(*

.. <legal notes>

legal notes
=================
| SPDX-FileCopyrightText: © 2026 Oleksandr Tiutyk <trofimich@gmail.com>
| SPDX-License-Identifier: LGPL-3.0-only
| For details check: LGPL-3.0-only_

.. _LGPL-3.0-only: https://www.gnu.org/licenses/lgpl-3.0.en.html

.. </legal notes>

*)

{attribute 'no_explicit_call' := 'do not call this function block directly'} 
FUNCTION_BLOCK SignalControlledIntersectionAutomationController EXTENDS TOF_Automation.AutomationController<7>
VAR CONSTANT
	RED_GREEN_LIGHT_INTERVAL : TIME := T#4000MS;
	YELLOW_LIGHT_INTERVAL : TIME := T#1000MS;
	FLASHING_YELLOW_LIGHT_INTERVAL : TIME := T#800MS;	
	
	SWITCH_SPEED_FACTOR : LREAL := 3; // +/- 30%
END_VAR
VAR_INPUT
	ThrowTestExceptionRequest : BOOL;
	TestExceptionMessage : STRING := 'Test error message';

	ResetRequest : BOOL;
END_VAR
VAR_OUTPUT	
	IntersectionMode : SIGNAL_CONTROLLED_INTERSECTION_MODE;
	IntersectionState : SIGNAL_CONTROLLED_INTERSECTION_STATE;

	{region "Devices"}
	
	WorkingModeSwitch : TOF_Devices_IO.DigitalInput("WorkingModeSwitch", THIS^);
	
	BlinkingYellowModeSwitch : TOF_Devices_IO.DigitalInput("BlinkingYellowModeSwitch", THIS^);
	
	SpeedAdjusterConverter : TOF_Devices_IO.RangeAnalogValueConverter(-20, +20, TOF_Devices_IO.RawAnalogValues.FromInt16(TOF_Core.SignedInt16.MIN_VALUE), TOF_Devices_IO.RawAnalogValues.FromInt16(TOF_Core.SignedInt16.MAX_VALUE));
	SwitchSpeedAdjuster : TOF_Devices_IO.AnalogInput("SwitchSpeedAdjuster", THIS^, SpeedAdjusterConverter);
	
	TrafficLight1 : TrafficLight("TrafficLight1", THIS^);
	TrafficLight2 : TrafficLight("TrafficLight2", THIS^);
	TrafficLight3 : TrafficLight("TrafficLight3", THIS^);
	TrafficLight4 : TrafficLight("TrafficLight4", THIS^);
	
 	{endregion} 	
END_VAR
VAR	
	_ClassName : STRING := __POUNAME();

	_Devices : ARRAY [0.._ChildCount - 1] OF TOF_Automation.IChildAutomationComponent := 
	[
		WorkingModeSwitch, 
		BlinkingYellowModeSwitch, 
		SwitchSpeedAdjuster, 
		TrafficLight1, 
		TrafficLight2, 
		TrafficLight3, 
		TrafficLight4
	];
	
	_OperationalStateChanged : BOOL;
	
	{region "Timers"}
	
	_RedGreenLightTimer : TOF_Timers.Timer;
	_YellowLightTimer : TOF_Timers.Timer;

	_FlashingYellowLightTimer : TOF_Timers.Timer;
	
	{endregion}
END_VAR

METHOD PRIVATE bindIO
WorkingModeSwitch.BindToIO(
	Terminals.DI_1.Channel_1
);

BlinkingYellowModeSwitch.BindToIO(
	Terminals.DI_1.Channel_2
);

SwitchSpeedAdjuster.BindToInt16IO(Terminals.AI_3.Channel_1);

TrafficLight1.BindToIO(
	redLightRawValue 	:= Terminals.DO_2.Channel_1,
	yellowLightRawValue := Terminals.DO_2.Channel_2,
	greenLightRawValue 	:= Terminals.DO_2.Channel_3	
);
TrafficLight2.BindToIO(
	redLightRawValue 	:= Terminals.DO_2.Channel_4,
	yellowLightRawValue := Terminals.DO_2.Channel_5,
	greenLightRawValue 	:= Terminals.DO_2.Channel_6	
);
TrafficLight3.BindToIO(
	redLightRawValue 	:= Terminals.DO_2.Channel_7,
	yellowLightRawValue := Terminals.DO_2.Channel_8,
	greenLightRawValue 	:= Terminals.DO_2.Channel_9	
);
TrafficLight4.BindToIO(
	redLightRawValue 	:= Terminals.DO_2.Channel_10,
	yellowLightRawValue := Terminals.DO_2.Channel_11,
	greenLightRawValue 	:= Terminals.DO_2.Channel_12	
);
END_METHOD

METHOD PRIVATE calculateCorrectedInterval : TIME
VAR_INPUT
	originalInterval : TIME;
	correctionPercent : SINT(-50..50);
END_VAR
IF correctionPercent = 0 THEN
	calculateCorrectedInterval := originalInterval;
ELSIF correctionPercent > 0 THEN
	calculateCorrectedInterval := originalInterval + TO_TIME(TO_INT(originalInterval) * correctionPercent / 100);
ELSE
	calculateCorrectedInterval := originalInterval - TO_TIME(TO_INT(originalInterval) * -correctionPercent / 100);
END_IF
END_METHOD

PROPERTY Children : REFERENCE TO ARRAY [0.._ChildCount - 1] OF TOF_Automation.IChildAutomationComponent
GET
Children REF= _Devices;
END_GET
END_PROPERTY

{attribute 'monitoring' := 'call'}
PROPERTY ClassName : STRING
GET
ClassName := _ClassName;
END_GET
END_PROPERTY

METHOD PRIVATE executeTimers
_RedGreenLightTimer.Execute();
_YellowLightTimer.Execute();
_FlashingYellowLightTimer.Execute();
END_METHOD

{attribute 'monitoring' := 'call'}
PROPERTY NamespaceName : STRING
GET
NamespaceName := CurrentNamespace.Name;
END_GET
END_PROPERTY

METHOD PROTECTED OnBeforeChildrenInitializing
_RedGreenLightTimer.Interval := RED_GREEN_LIGHT_INTERVAL;
_YellowLightTimer.Interval := YELLOW_LIGHT_INTERVAL;

_FlashingYellowLightTimer.Interval := FLASHING_YELLOW_LIGHT_INTERVAL;

bindIO();
END_METHOD

METHOD PROTECTED OnFault
startIdelingMode();

IF ResetRequest THEN
	ResetRequest := FALSE;
	
	Reset();
END_IF
END_METHOD

METHOD PROTECTED OnOperationalStateChanged
VAR_INPUT
	previousState : TOF_Automation.OPERATIONAL_STATE;
END_VAR
_OperationalStateChanged := TRUE;
END_METHOD

METHOD PROTECTED OnWorking
VAR
	testException : TOF_Core.StandardException;
END_VAR
executeTimers();

IF _OperationalStateChanged OR_ELSE WorkingModeSwitch.Changed OR_ELSE BlinkingYellowModeSwitch.Changed THEN
	_OperationalStateChanged := FALSE;
	
	IF NOT WorkingModeSwitch.Value THEN
		startIdelingMode();
	ELSE
		IF BlinkingYellowModeSwitch.Value THEN
			startBlinkingYellowMode();
		ELSE
			startNormalMode();
		END_IF	
	END_IF
	
	RETURN;
ELSE
	CASE IntersectionMode OF
		SIGNAL_CONTROLLED_INTERSECTION_MODE.NORMAL:
			processNormalMode();
		
		SIGNAL_CONTROLLED_INTERSECTION_MODE.BLINKING_YELLOW:
			processBlinkingYellowMode();
	END_CASE
END_IF

IF ThrowTestExceptionRequest THEN
	ThrowTestExceptionRequest := FALSE;
	testException.ThrowByObject(THIS^, __POUNAME(), __POSITION(), TO_WSTRING(TestExceptionMessage), 0);
END_IF
END_METHOD

{attribute 'monitoring' := 'call'}
PROPERTY OperationalStateName : STRING(16)
GET
OperationalStateName := TO_STRING(_OperationalState);
END_GET
END_PROPERTY

METHOD PRIVATE processBlinkingYellowMode
IF _FlashingYellowLightTimer.Elapsed THEN
	IF IntersectionState = SIGNAL_CONTROLLED_INTERSECTION_STATE.ALL_YELLOW THEN
		IntersectionState := SIGNAL_CONTROLLED_INTERSECTION_STATE.ALL_OFF;
	ELSE
		IntersectionState := SIGNAL_CONTROLLED_INTERSECTION_STATE.ALL_YELLOW;
	END_IF
	
	startFlashingYellowLightTimer();
	
	updateTraficLights();
END_IF
END_METHOD

METHOD processNormalMode
CASE IntersectionState OF
	SIGNAL_CONTROLLED_INTERSECTION_STATE._1_3_GREEN_AND_2_4_RED:
		IF _RedGreenLightTimer.Elapsed THEN
			startYellowLightTimer();
			IntersectionState := SIGNAL_CONTROLLED_INTERSECTION_STATE._1_3_YELLOW_AND_2_4_YELLOW;
			updateTraficLights();
		END_IF
 
	SIGNAL_CONTROLLED_INTERSECTION_STATE._1_3_YELLOW_AND_2_4_YELLOW:
		IF _YellowLightTimer.Elapsed THEN
			startRedGreenLightTimer();
			IntersectionState := SIGNAL_CONTROLLED_INTERSECTION_STATE._2_4_GREEN_AND_1_3_RED;
			updateTraficLights();
		END_IF
	
	SIGNAL_CONTROLLED_INTERSECTION_STATE._2_4_GREEN_AND_1_3_RED:
		IF _RedGreenLightTimer.Elapsed THEN
			startYellowLightTimer();
			IntersectionState := SIGNAL_CONTROLLED_INTERSECTION_STATE._2_4_YELLOW_AND_1_3_YELLOW;
			updateTraficLights();
		END_IF
	
	SIGNAL_CONTROLLED_INTERSECTION_STATE._2_4_YELLOW_AND_1_3_YELLOW:
		IF _YellowLightTimer.Elapsed THEN
			startRedGreenLightTimer();
			IntersectionState := SIGNAL_CONTROLLED_INTERSECTION_STATE._1_3_GREEN_AND_2_4_RED;
			updateTraficLights();
		END_IF
	
	ELSE
		startRedGreenLightTimer();
		IntersectionState := SIGNAL_CONTROLLED_INTERSECTION_STATE._1_3_GREEN_AND_2_4_RED;
		updateTraficLights();
END_CASE
END_METHOD

{attribute 'monitoring' := 'call'}
PROPERTY SelfSize : ULINT
GET
SelfSize := XSIZEOF(THIS^);
END_GET
END_PROPERTY

METHOD PRIVATE startBlinkingYellowMode
_RedGreenLightTimer.Cancel();
_YellowLightTimer.Cancel();

startFlashingYellowLightTimer();

IntersectionMode := SIGNAL_CONTROLLED_INTERSECTION_MODE.BLINKING_YELLOW;
IntersectionState := SIGNAL_CONTROLLED_INTERSECTION_STATE.ALL_YELLOW;

updateTraficLights();
END_METHOD

METHOD PRIVATE startFlashingYellowLightTimer
_FlashingYellowLightTimer.Interval := calculateCorrectedInterval(FLASHING_YELLOW_LIGHT_INTERVAL, TO_SINT(SWITCH_SPEED_FACTOR * SwitchSpeedAdjuster.Value));

_FlashingYellowLightTimer.Restart();
END_METHOD

METHOD startIdelingMode
_RedGreenLightTimer.Cancel();
_YellowLightTimer.Cancel();
_FlashingYellowLightTimer.Cancel();

IntersectionMode := SIGNAL_CONTROLLED_INTERSECTION_MODE.IDELING;
IntersectionState := SIGNAL_CONTROLLED_INTERSECTION_STATE.ALL_OFF;

updateTraficLights();
END_METHOD

METHOD startNormalMode
startRedGreenLightTimer();

_YellowLightTimer.Cancel();
_FlashingYellowLightTimer.Cancel();

IntersectionMode := SIGNAL_CONTROLLED_INTERSECTION_MODE.NORMAL;
IntersectionState := SIGNAL_CONTROLLED_INTERSECTION_STATE._1_3_GREEN_AND_2_4_RED;

updateTraficLights();
END_METHOD

METHOD PRIVATE startRedGreenLightTimer
_RedGreenLightTimer.Interval := calculateCorrectedInterval(RED_GREEN_LIGHT_INTERVAL, TO_SINT(SWITCH_SPEED_FACTOR * SwitchSpeedAdjuster.Value));

_RedGreenLightTimer.Restart();
END_METHOD

METHOD PRIVATE startYellowLightTimer
_YellowLightTimer.Interval := calculateCorrectedInterval(YELLOW_LIGHT_INTERVAL, TO_SINT(SWITCH_SPEED_FACTOR * SwitchSpeedAdjuster.Value));

_YellowLightTimer.Restart();
END_METHOD

METHOD PRIVATE updateTraficLights
CASE IntersectionState OF
	SIGNAL_CONTROLLED_INTERSECTION_STATE.ALL_OFF:
		TrafficLight1.SetLight(TRAFFIC_LIGHT_COLOR.NO_COLOR);
		TrafficLight2.SetLight(TRAFFIC_LIGHT_COLOR.NO_COLOR);
		TrafficLight3.SetLight(TRAFFIC_LIGHT_COLOR.NO_COLOR);
		TrafficLight4.SetLight(TRAFFIC_LIGHT_COLOR.NO_COLOR);
	
	SIGNAL_CONTROLLED_INTERSECTION_STATE.ALL_YELLOW, 
	SIGNAL_CONTROLLED_INTERSECTION_STATE._1_3_YELLOW_AND_2_4_YELLOW,
	SIGNAL_CONTROLLED_INTERSECTION_STATE._2_4_YELLOW_AND_1_3_YELLOW:
		TrafficLight1.SetLight(TRAFFIC_LIGHT_COLOR.YELLOW);
		TrafficLight2.SetLight(TRAFFIC_LIGHT_COLOR.YELLOW);
		TrafficLight3.SetLight(TRAFFIC_LIGHT_COLOR.YELLOW);
		TrafficLight4.SetLight(TRAFFIC_LIGHT_COLOR.YELLOW);
	
	SIGNAL_CONTROLLED_INTERSECTION_STATE._1_3_GREEN_AND_2_4_RED:
		TrafficLight1.SetLight(TRAFFIC_LIGHT_COLOR.GREEN);
		TrafficLight2.SetLight(TRAFFIC_LIGHT_COLOR.RED);
		TrafficLight3.SetLight(TRAFFIC_LIGHT_COLOR.GREEN);
		TrafficLight4.SetLight(TRAFFIC_LIGHT_COLOR.RED);
	
	SIGNAL_CONTROLLED_INTERSECTION_STATE._2_4_GREEN_AND_1_3_RED:
		TrafficLight1.SetLight(TRAFFIC_LIGHT_COLOR.RED);
		TrafficLight2.SetLight(TRAFFIC_LIGHT_COLOR.GREEN);
		TrafficLight3.SetLight(TRAFFIC_LIGHT_COLOR.RED);
		TrafficLight4.SetLight(TRAFFIC_LIGHT_COLOR.GREEN);
END_CASE
END_METHOD

END_FUNCTION_BLOCK

(* stored: Version 1.1.0.1
   POU SignalControlledIntersectionAutomationController: Id {d0f0aa39-ea76-461a-8fa3-dba15b8635a6}, SpecialFunc None
   Folder Overriden methods: Id {13702960-9d99-4885-a6ce-63462aae1b07}
   Folder Service methods: Id {856d71ee-39f1-4125-9914-d1908aaa9de4}
   Folder Process mode: Id {9df05ec4-b756-4783-a76b-40e885978be7}
   Folder Start mode: Id {5736814f-405d-4520-8342-b8d268de143f}
   Folder Start timer: Id {c16a13e4-4c94-4831-b2dc-b8960e14f551}
   Method bindIO: Id {1bc433ca-8d0e-4452-8e3c-75449de42a8a}
   Method calculateCorrectedInterval: Id {51d751ca-80fc-4362-91e8-31296f350aff}
   Property Children: Id {edb09d7e-eaa4-4ee7-bf71-f499880b4098}
   Get Get: Id {90a76f6a-9caa-4ca6-88e8-931aff742de9}
   Property ClassName: Id {533645c9-51ab-4278-b915-2be070529db7}
   Get Get: Id {1aae8f98-7140-4915-9ec0-3cdf6e26caf7}
   Method executeTimers: Id {dfed4c3f-27bc-4f55-8a83-85a2d79b2492}
   Property NamespaceName: Id {b7a7d419-b6f1-4dfe-b4b4-ae9ac4b21e47}
   Get Get: Id {225fc0aa-c40a-4b1c-a5e5-ec5ea749c036}
   Method OnBeforeChildrenInitializing: Id {d14266f5-308f-4ec2-bbd3-dd4787db6449}
   Method OnFault: Id {6fcc8089-8d26-4d23-ab84-876516fe47cb}
   Method OnOperationalStateChanged: Id {dfa58b81-4624-4688-b85b-fa55f112c836}
   Method OnWorking: Id {89569639-43c3-4fe5-81a2-97d1904a242b}
   Property OperationalStateName: Id {af99d547-78da-4f00-96bd-32d0d0304681}
   Get Get: Id {7a068cfa-95a9-4134-b604-ea1c07f183d2}
   Method processBlinkingYellowMode: Id {62fb35a3-197f-483b-a168-1d68d2c02c71}
   Method processNormalMode: Id {a778b296-2e19-469e-8475-30ab670a6dcd}
   Property SelfSize: Id {db85e590-8997-4b56-bd9a-8e5dd4df70fe}
   Get Get: Id {f6ab4eca-dad6-4656-bd85-433d2bf1854b}
   Method startBlinkingYellowMode: Id {338031f0-6ea3-4eea-a4fb-410b4cc13072}
   Method startFlashingYellowLightTimer: Id {96309d45-677b-4977-9f1c-e21c0143efbb}
   Method startIdelingMode: Id {8ddb5609-6544-4dcc-b972-500abb23f0f5}
   Method startNormalMode: Id {bfa9afc6-d6b0-4dbc-b2b3-10d6e8a939c6}
   Method startRedGreenLightTimer: Id {50f36714-64fe-4212-afb9-2e8a39734cfd}
   Method startYellowLightTimer: Id {75f70f4d-af10-457d-91be-f1022c3b5646}
   Method updateTraficLights: Id {f60cca55-65f4-4222-8c1f-0c67e0a9c589} *)
